(* PLC project liner_cyclic.project, CODESYS CODESYS V3.5 SP17 Patch 3 *)
(* stored: creationDateTime 1970-01-01T00:00:00, modificationDateTime 1970-01-01T00:00:00 *)

FUNCTION_BLOCK LinearSensorHandle
  VAR_INPUT
    position : UDINT;
  END_VAR
  VAR_OUTPUT
    Calc_position_mm : REAL;
  END_VAR
  VAR
    tmp : REAL;
  END_VAR

            tmp := UDINT_TO_REAL(position);
Calc_position_mm := tmp / 1000; 

          
END_FUNCTION_BLOCK
